{attribute 'linkalways'} 
{attribute 'no_explicit_call' := 'This FB is a CLASS and must be accessed using methods or properties'}
{attribute 'enable_dynamic_creation'}
FUNCTION_BLOCK Dictionary EXTENDS Disposable IMPLEMENTS I_Dictionary
VAR
	eventEmitter : EventEmitter;
	rootNode : I_DictionaryTreeNode;
END_VAR

METHOD PUBLIC AddOrUpdate
VAR_INPUT
	Key : T_MAXSTRING;
	Value : ANY;
END_VAR
rootNode := THIS^.RecursiveInsert(Key, Value, rootNode);
EmitChangedEvent();
END_METHOD

METHOD PRIVATE Balance : I_DictionaryTreeNode
VAR_INPUT
	Node : I_DictionaryTreeNode;
END_VAR
VAR
	balanceFactor : DINT;
END_VAR
balanceFactor := THIS^.GetBalanceFactor(Node);

IF (balanceFactor > 1) THEN
	IF THIS^.GetBalanceFactor(Node.Left) < 0 THEN
		Node.Left := THIS^.LeftRotate(Node.Left);
	END_IF
	Node := RightRotate(Node);
ELSIF (balanceFactor < -1) THEN
	IF THIS^.GetBalanceFactor(Node.Right) > 0 THEN
		Node.Right := RightRotate(Node.Right);
	END_IF
	Node := LeftRotate(Node);
END_IF

Balance := Node;
END_METHOD

METHOD PUBLIC Clear
VAR_INPUT
END_VAR
IF rootNode = 0 THEN
	RETURN;
END_IF

THIS^.RecursiveClear(rootNode);
rootNode := 0;
EmitChangedEvent();
END_METHOD

METHOD PUBLIC ContainsKey : BOOL
VAR_INPUT
	Key : T_MAXSTRING;
END_VAR
VAR
	foundNode : I_DictionaryTreeNode;
END_VAR
foundNode := THIS^.RecursiveFind(Key, rootNode);

IF foundNode = 0 THEN
	RETURN;
END_IF

ContainsKey := TRUE;
END_METHOD

PROPERTY PUBLIC Count : DINT
GET
VAR
	NodeCount : DINT;
END_VAR
RecursiveCountNodes(rootNode, NodeCount);
Count := NodeCount;
END_GET
END_PROPERTY

METHOD PRIVATE EmitChangedEvent
VAR
	pDictionaryChangedEvent : POINTER TO KeyValueCollectionChangedEvent;
END_VAR
pDictionaryChangedEvent := __NEW(KeyValueCollectionChangedEvent(Target := THIS^));
eventEmitter.Emit('OnChanged', pDictionaryChangedEvent^);
pDictionaryChangedEvent^.Dispose();
END_METHOD

METHOD PRIVATE EmitDisposedEvent
VAR
	pDictionaryDisposedEvent : POINTER TO KeyValueCollectionDisposedEvent;
END_VAR
pDictionaryDisposedEvent := __NEW(KeyValueCollectionDisposedEvent(Target := THIS^));
eventEmitter.Emit('OnDisposed', pDictionaryDisposedEvent^);
pDictionaryDisposedEvent^.Dispose();
END_METHOD

METHOD FB_exit : BOOL
VAR_INPUT
	bInCopyCode : BOOL; // if TRUE, the exit method is called for exiting an instance that is copied afterwards (online change).
END_VAR
VAR
END_VAR
IF bInCopyCode THEN
    RETURN;
END_IF

Clear();
EmitDisposedEvent();
END_METHOD

METHOD PRIVATE FindMinimum : I_DictionaryTreeNode
VAR_INPUT
	Node : I_DictionaryTreeNode;
END_VAR
VAR
	nextNode : I_DictionaryTreeNode;
END_VAR
nextNode := Node;

WHILE (nextNode.left <> 0) DO
      nextNode := nextNode.left;
END_WHILE;

FindMinimum := nextNode;
END_METHOD

METHOD PRIVATE GetBalanceFactor : DINT
VAR_INPUT
	Node : I_DictionaryTreeNode;
END_VAR
IF (Node = 0) THEN
	GetBalanceFactor := 0;
	RETURN;
END_IF

GetBalanceFactor := THIS^.GetHeight(node.left) - THIS^.GetHeight(node.right);
END_METHOD

METHOD GetEnumerator : I_ForwardEnumerator
VAR
	pNodeCollection : POINTER TO LinkedList;
	pEnumerator : POINTER TO DictionaryForwardEnumerator;
END_VAR
pNodeCollection := __NEW(LinkedList);
THIS^.RecursiveAddNodesInOrderToCollection(rootNode, pNodeCollection^);

pEnumerator := __NEW(DictionaryForwardEnumerator(Parent := THIS^, Nodes := pNodeCollection^));
GetEnumerator := pEnumerator^;
END_METHOD

METHOD PRIVATE GetHeight : DINT
VAR_INPUT
	Node : I_DictionaryTreeNode;
END_VAR
IF Node = 0 THEN
	GetHeight := -1;
	RETURN;
END_IF

GetHeight := Node.Height;
END_METHOD

METHOD PUBLIC GetKeys : I_Collection
VAR
	pLinkedList : POINTER TO LinkedList;
END_VAR
pLinkedList := __NEW(LinkedList);
THIS^.RecursiveAddKeysInOrderToCollection(rootNode,pLinkedList^);
GetKeys := pLinkedList^;
END_METHOD

METHOD GetKeyValueEnumerator : I_KeyValueForwardEnumerator
VAR
	pNodeCollection : POINTER TO LinkedList;
	pEnumerator : POINTER TO DictionaryForwardEnumerator;
END_VAR
pNodeCollection := __NEW(LinkedList);
THIS^.RecursiveAddNodesInOrderToCollection(rootNode, pNodeCollection^);

pEnumerator := __NEW(DictionaryForwardEnumerator(Parent := THIS^, Nodes := pNodeCollection^));
GetKeyValueEnumerator := pEnumerator^;
END_METHOD

PROPERTY IsEmpty : BOOL
GET
IsEmpty := rootNode = 0;
END_GET
END_PROPERTY

METHOD PRIVATE LeftRotate : I_DictionaryTreeNode
VAR_INPUT
	X : I_DictionaryTreeNode;
END_VAR
VAR
	y : I_DictionaryTreeNode;
	t2 : I_DictionaryTreeNode;
END_VAR
y := X.right;
t2 := y.left;
y.left := X;
X.right := t2;
THIS^.UpdateHeight(X);
THIS^.UpdateHeight(y);
LeftRotate := y;
END_METHOD

METHOD PUBLIC OffEvent
VAR_INPUT
	EventName : T_MaxString;
	EventHandler : I_EventHandler;
END_VAR
eventEmitter.OffEvent(EventName, EventHandler);
END_METHOD

METHOD PUBLIC OnceEvent
VAR_INPUT
	EventName : T_MaxString;
	EventHandler : I_EventHandler;
END_VAR
eventEmitter.OnceEvent(EventName, EventHandler);
END_METHOD

METHOD PUBLIC OnEvent
VAR_INPUT
	EventName : T_MaxString;
	EventHandler : I_EventHandler;
END_VAR
eventEmitter.OnEvent(EventName, EventHandler);
END_METHOD

METHOD PRIVATE RecursiveAddKeysInOrderToCollection
VAR_INPUT
	Node : I_DictionaryTreeNode;
	Collection : I_Collection;
END_VAR
VAR
	key : T_MAXSTRING;
END_VAR
IF Node = 0 THEN
	RETURN;
END_IF

THIS^.RecursiveAddKeysInOrderToCollection(Node.Left,Collection);
key := Node.Key;
Collection.AddItem(key);
THIS^.RecursiveAddKeysInOrderToCollection(Node.Right,Collection);
END_METHOD

METHOD PRIVATE RecursiveAddNodesInOrderToCollection
VAR_INPUT
	Node : I_DictionaryTreeNode;
	Collection : I_Collection;
END_VAR
IF Node = 0 THEN
	RETURN;
END_IF

THIS^.RecursiveAddNodesInOrderToCollection(Node.Left,Collection);
Collection.AddItem(Node);
THIS^.RecursiveAddNodesInOrderToCollection(Node.Right,Collection);
END_METHOD

METHOD PRIVATE RecursiveClear
VAR_INPUT
	Node : I_DictionaryTreeNode;
END_VAR
VAR
	thisNodeKey : T_MAXSTRING;
	leftNodeKey : T_MAXSTRING;
	rightNodeKey : T_MAXSTRING;
END_VAR
IF (Node = 0) THEN
	RETURN;
END_IF

thisNodeKey := Node.key;

IF (Node.Left <> 0) THEN
	leftNodeKey := Node.Left.key;
END_IF

IF (Node.Right <> 0) THEN
	rightNodeKey := Node.Right.key;
END_IF


RecursiveClear(Node.Left);
RecursiveClear(Node.Right);
Node.Dispose();
END_METHOD

METHOD PRIVATE RecursiveCountNodes
VAR_INPUT
	Node : I_DictionaryTreeNode;
	Count : REFERENCE TO DINT;
END_VAR
IF Node = 0 THEN
	RETURN;
END_IF

Count := Count + 1;

THIS^.RecursiveCountNodes(Node.Left,Count);
THIS^.RecursiveCountNodes(Node.Right,Count);
END_METHOD

METHOD PRIVATE RecursiveDelete : I_DictionaryTreeNode
VAR_INPUT
	Key : T_MAXSTRING;
	Node : I_DictionaryTreeNode;
END_VAR
VAR
	newNode : I_DictionaryTreeNode; 
	minValueNode : I_DictionaryTreeNode;
	minValueNodeParent : I_DictionaryTreeNode;
	balanceFactor : DINT;
END_VAR
IF (Node = 0) THEN
    RETURN;
END_IF

IF (Key < Node.Key) THEN
    Node.left := THIS^.RecursiveDelete(Key, Node.left);
ELSIF (Key > Node.Key) THEN
    Node.right := THIS^.RecursiveDelete(Key, Node.right);
ELSE
    IF (Node.Left = 0) OR (Node.Right = 0) THEN
        IF (Node.Left = 0) THEN
            newNode := Node.Right;
        ELSE
            newNode := Node.Left;
        END_IF

        Node.Dispose();
        THIS^.updateHeight(newNode);
        RecursiveDelete := THIS^.Balance(newNode);
        RETURN;
    ELSE
        minValueNode := FindMinimum(Node.Right);
        Node.Clone(minValueNode);
        Node.Right := THIS^.RecursiveDelete(minValueNode.Key, Node.Right);	
    END_IF
END_IF

THIS^.updateHeight(Node);
RecursiveDelete := THIS^.Balance(Node);
END_METHOD

METHOD PRIVATE RecursiveFind : I_DictionaryTreeNode
VAR_INPUT
	Key : T_MAXSTRING;
	Node : I_DictionaryTreeNode;
END_VAR
IF (Node = 0) THEN
	RETURN;
END_IF

IF (Key < Node.key) THEN
  RecursiveFind := THIS^.RecursiveFind(key, Node.left);
  RETURN;
ELSIF (key > Node.key) THEN
  RecursiveFind := THIS^.RecursiveFind(key, Node.right);
  RETURN;
ELSE 
  RecursiveFind := Node;
  RETURN;
END_IF
END_METHOD

METHOD PRIVATE RecursiveInsert : I_DictionaryTreeNode
VAR_INPUT
	Key : T_MAXSTRING;
	Value : ANY;
	Node : I_DictionaryTreeNode;
END_VAR
VAR
	pAVLTreeNode : POINTER TO DictionaryTreeNode;
	balanceFactor : DINT;
END_VAR
IF (Node = 0) THEN
	pAVLTreeNode := __NEW(DictionaryTreeNode(NodeKey := Key, NodeSource := Value));
	RecursiveInsert := pAVLTreeNode^;
	RETURN;
END_IF

IF (Key < Node.Key) THEN
	Node.left := THIS^.RecursiveInsert(Key, Value, Node.left);
ELSIF (Key > Node.Key) THEN
	Node.right := THIS^.RecursiveInsert(Key, Value, Node.right);
ELSE
	Node.Reinitialize(Key,Value);
	RecursiveInsert := Node;
END_IF

THIS^.updateHeight(node);

balanceFactor := THIS^.GetBalanceFactor(Node);
Node := balance(Node);
RecursiveInsert := Node;
END_METHOD

METHOD PUBLIC Remove
VAR_INPUT
	Key : T_MAXSTRING;
END_VAR
rootNode := THIS^.RecursiveDelete(Key, rootNode);
EmitChangedEvent();
END_METHOD

METHOD PRIVATE RightRotate : I_DictionaryTreeNode
VAR_INPUT
	Y : I_DictionaryTreeNode;
END_VAR
VAR
	x : I_DictionaryTreeNode;
	t2 : I_DictionaryTreeNode;
END_VAR
x := Y.left;
t2 := x.right;
x.right := Y;
Y.left := t2;
THIS^.UpdateHeight(Y);
THIS^.UpdateHeight(x);
RightRotate := x;
END_METHOD

METHOD PUBLIC TryAdd : BOOL
VAR_INPUT
	Key : T_MAXSTRING;
	Value : ANY;
END_VAR
IF ContainsKey(Key) THEN
	RETURN;
END_IF
	  
THIS^.AddOrUpdate(Key, Value);
TryAdd := TRUE;
END_METHOD

METHOD PUBLIC TryGetValue : BOOL
VAR_INPUT
	Key : T_MAXSTRING;
	Destination	: ANY;
END_VAR
TryGetValue := TryGetValueTo(Key, Destination.pValue, DINT_TO_UDINT(Destination.diSize));
END_METHOD

METHOD PUBLIC TryGetValueTo : BOOL
VAR_INPUT
	Key : T_MAXSTRING;
	DestinationAddress : PVOID;
	DestinationSize : UDINT;
END_VAR
VAR
	foundNode : I_DictionaryTreeNode;
END_VAR
foundNode := THIS^.RecursiveFind(Key, rootNode);

IF foundNode = 0 THEN
	RETURN;
END_IF

TryGetValueTo := foundNode.TryGetTo(DestinationAddress, DestinationSize);
END_METHOD

METHOD PRIVATE UpdateHeight
VAR_INPUT
	Node : I_DictionaryTreeNode;
END_VAR
IF (Node = 0) THEN
	RETURN;
END_IF

Node.height := 1 + MAX(THIS^.GetHeight(Node.left), THIS^.GetHeight(Node.right));
END_METHOD

END_FUNCTION_BLOCK

(* stored: Version 1.1.0.1, ProductVersion 3.1.4024.12
   POU Dictionary: Id {fecf5b10-b0d6-0a2e-0b01-2d74663542c7}, SpecialFunc None
   Folder Destructor: Id {eed191c7-3b43-0817-3c1e-383a024a4a99}
   Folder Private: Id {92854147-ba41-0344-0d9a-013335b79904}
   Method AddOrUpdate: Id {ece2ca9c-a079-0658-3d4a-24912afdb3a4}
   Method Balance: Id {84e8670a-47b6-0fa0-333c-26a7475d8ca7}
   Method Clear: Id {a6201ffe-9631-0ef2-3fe4-e47ac785e7a2}
   Method ContainsKey: Id {3d74f456-d7df-07d9-2989-070f70587903}
   Property Count: Id {10d90968-c8e5-0865-21d6-fc82dc2ab1ae}
   Get Get: Id {cd6ace64-5417-0720-0881-b4c0dd96efd6}
   Method EmitChangedEvent: Id {a9b49c43-111a-09b6-1239-623bb33f1048}
   Method EmitDisposedEvent: Id {91ef6ef7-e417-0fe2-0875-0585ae579942}
   Method FB_exit: Id {3e757861-735f-0920-2778-50722bd1e0c6}
   Method FindMinimum: Id {fc2ea284-32ce-016c-361c-c2eae2a03949}
   Method GetBalanceFactor: Id {24138e83-e253-0881-3f13-e45ac736c7ae}
   Method GetEnumerator: Id {294054ea-4a41-02aa-097a-eee4c2d5c2a0}
   Method GetHeight: Id {018a9014-719c-020c-2bc5-73af29fda4ac}
   Method GetKeys: Id {c5c6bed8-1459-0ffc-0dfd-f6b3e29c5d97}
   Method GetKeyValueEnumerator: Id {da2ced37-a2f7-0246-0970-72e95bfcb69d}
   Property IsEmpty: Id {ec628771-b0f1-04dd-3b54-e19571091848}
   Get Get: Id {7f5cb21e-a6f4-0c98-0aff-d044a36317c4}
   Method LeftRotate: Id {7998d758-83d1-0816-1fa0-c9acda7c1bc7}
   Method OffEvent: Id {a014b525-9ff5-0b8a-1ead-fa954b6bca8f}
   Method OnceEvent: Id {914215dd-ec5d-0eae-126a-b10b5a76b958}
   Method OnEvent: Id {c8c48b54-f04b-0e1e-0048-be0a2caf5dec}
   Method RecursiveAddKeysInOrderToCollection: Id {ace22016-259d-0957-1de1-b25b2ad387f1}
   Method RecursiveAddNodesInOrderToCollection: Id {09d61aa0-73bf-076a-19c2-2cafbe84f84b}
   Method RecursiveClear: Id {a4f868c3-ad4b-0f06-20eb-496818387d2c}
   Method RecursiveCountNodes: Id {08299698-30d8-05a2-1af2-fc132107a98c}
   Method RecursiveDelete: Id {6b4f87c5-b2b3-0877-196e-621c2c7648a6}
   Method RecursiveFind: Id {61c91ed6-ee61-09d3-103f-f866f6c22531}
   Method RecursiveInsert: Id {107a9424-354b-055f-031a-f471a79b1581}
   Method Remove: Id {59e40474-4182-0ecf-3bfb-32ab2df562ad}
   Method RightRotate: Id {caffc819-b202-0f61-282a-29f2d7b19cca}
   Method TryAdd: Id {2e702fe5-a018-01b2-12e4-5390fc008087}
   Method TryGetValue: Id {55a3c8b0-17de-0463-147a-468a6592f8ac}
   Method TryGetValueTo: Id {13ca6bb5-5fb6-0903-2dd7-30e5c4632b54}
   Method UpdateHeight: Id {a5f839b3-5e38-011d-0faf-1c3ff19a72aa} *)
